// TIA Portal V20 export
DATA_BLOCK "instFB_TeachCtrl"   // DB28
VERSION : 1.1
// Instance DB for FB_TeachCtrl V1.0 (Module F, 2026-05-23). 7 R_TRIG edge detectors (Capture, Verify, Clear, ClearAll, StartReplay, StopReplay, MoveDone) + statTeachOK gate. FB writes to shared GDB_AxisCtrl.LKinCtrl.input.{jogframe, movelinear} - no local MC instance.
// stored: InstanceOfName FB_TeachCtrl, InstanceOfType FB
"FB_TeachCtrl"
   // VAR
   //    sRTRIG_Capture { S7_SetPoint := 'True'} : R_TRIG;
   //    sRTRIG_Verify { S7_SetPoint := 'True'} : R_TRIG;
   //    sRTRIG_Clear { S7_SetPoint := 'True'} : R_TRIG;
   //    sRTRIG_ClearAll { S7_SetPoint := 'True'} : R_TRIG;
   //    sRTRIG_StartReplay { S7_SetPoint := 'True'} : R_TRIG;
   //    sRTRIG_StopReplay { S7_SetPoint := 'True'} : R_TRIG;
   //    sRTRIG_MoveDone { S7_SetPoint := 'True'} : R_TRIG;
   //    statTeachOK : Bool;
   // END_VAR
BEGIN
END_DATA_BLOCK
